# B&R Automation Studio project perfxxl (part 2)

### motorfunc.h
```c
/*
                             *******************
******************************* C HEADER FILE *******************************
**                           *******************                           **
**                                                                         **
** project  : LS JET II                                                    **
** filename : MOTORFUNC.H                                                  **
** version  : 1.02                                                         **
** date     : 24.01.2008                                                   **
**                                                                         **
*****************************************************************************
** Abstract                                                                **
** ========                                                                **
** Declares the functions for motor control functions  	                   **
**                                                                         **
**                                                                         **
** Copyright (c) 2006, Krause-Biagosch GmbH                                **
** All rights reserved.                                                    **
**                                                                         **
*****************************************************************************
VERSION HISTORY:
----------------
Version     : 1.00
Date        : 20.10.2006
Revised by  : Herbert Aden
Description : Original version.

Version     : 1.01
Date        : 12.10.2007
Revised by  : Herbert Aden
Description : signature of MoveToAbsPosition has changed

Version     : 1.02
Date        : 24.01.2008
Revised by  : Herbert Aden
Description : Added define for ANSW0 command

*/

#ifndef _MOTORFUNC_INCLUDED
#define _MOTORFUNC_INCLUDED

/****************************************************************************/
/**                                                                        **/
/**                           INCLUDE FILES                                **/
/**                                                                        **/
/****************************************************************************/
/* NONE */

/****************************************************************************/
/**                                                                        **/
/**                       DEFINITIONS AND MACROS                           **/
/**                                                                        **/
/****************************************************************************/
#define CMDSTRINGLENGTH        (10)
#define DONT_SEND_SPEED        (0L)

#define CMD_RELATIVE_POS            "LR"
#define CMD_ABSOLUTE_POS            "LA"
#define CMD_SPEED                   "SP"
#define CMD_START_MOTION            "M"
#define CMD_CONT_CURRENT            "LCC"
#define CMD_PEAK_CURRENT            "LPC"
#define CMD_STOP                    "V0"
#define CMD_MOVE_AT                 "V"
/* for reference */
#define CMD_HOME                    "HO"
#define CMD_ENABLE                  "EN"
#define CMD_SERIAL                  "SOR0"
#define CMD_ACCELERATION            "AC"
#define CMD_PROPFACT                "POR"
#define CMD_INTFACT                 "I"
#define CMD_NOANSW                  "ANSW0"
#define CMD_COMPATIBLE              "COMPATIBLE1"

#define CMD_GETTEMP                 "TEM"
#define CMD_GETFAULTSTAT            "GFS"

/****************************************************************************/
/**                                                                        **/
/**                      TYPEDEFS AND STRUCTURES                           **/
/**                                                                        **/
/****************************************************************************/
typedef struct
{
	STRING	CmdString[CMDSTRINGLENGTH];  /* command string*/
	DINT	Parameter;          /* Parameter for the command */
	BOOL	UseParameter;       /* if true, the parameter is added to the command
	                             *  else the parameter is ignored
	                             */
	BOOL	UseRefDirection;    /* if true, the ref direction of the motor is used
	                             * to determine the direction of movement
	                             * hence the sign of parameter is irrelevant;
	                             * else the sign is used to determine direction
	                             */
	INT     SendMotor;          /* the motor which shall receive the command*/
	BOOL	Send;               /* the actual send command, stay TRUE until
	                             * sending finished
	                             */
	BOOL	Request;            /* indicates that data is requested from motor */
}SerialCmd_Typ;

/****************************************************************************/
/**                                                                        **/
/**                      EXPORTED VARIABLES                                **/
/**                                                                        **/
/****************************************************************************/
#ifndef _MOTORFUNC_C_SRC
extern _GLOBAL SerialCmd_Typ SerialCmd;
#endif

/****************************************************************************/
/**                                                                        **/
/**                          EXPORTED FUNCTIONS                            **/
/**                                                                        **/
/****************************************************************************/

/****************************************************************************/
/** Send commands to a motor                                                */
/****************************************************************************/
/**
 * Sends commands to a specified motor.
 * Example: Call MotorCmd(1,"LA",TRUE,200000)
 *          will send "1LA200000" to the interface
 *
 * Parameters: UINT  Motor        the motor to which the command is being sent
 *             char *CmdString    the command string (NULL terminated)
 *             BOOL  UseValue     if true, then the value will be added to the
 *                                command
 *             DINT  Value        the value to be added to the command
 *
 * Returns:    OK                 when finished sending
 *             NOT_OK             while waiting for sending
 *
**/
BOOL	SendMotorCmd(const INT pMotor,const char *CmdStr,const BOOL UseValue,const DINT Value);

/****************************************************************************/
/** Check, if a motor is in a certain position window                       */
/****************************************************************************/
/**
 * Checks, if the position of the specified motor is in a specified range
 * (Position window)
 * Example call: PositionOk(1,200000,100)
 *               returns false, as long as the motorposition is <199900
 *                                                           or >200100
 * Parameters: UINT  Motor        the motor to be checked
 *             DINT  Pos          the position where the motor should be
 *             DINT  Deviation    the maximum tolerated deviaition (+/-)
 *
 *
 * Returns:    OK                 if current motor position is in range
 *             NOT_OK             if current motor position is out of range
 *
**/
BOOL	isPositionOk(const INT Motor,DINT Pos,DINT Deviation)/*@modifies nothing@*/;

/****************************************************************************/
/** Check, if a motor is below a certain position                           */
/****************************************************************************/
/**
 * Checks, if the position of the specified motor is below a specified position
 * ATTENTION: Does not work, if actual position has a different sign than the
 *            given max position! May only be used with all positive or all negative
 *            values. E.g. if the atual position is 1000 and we test for -1000 the
 *            function will return true, which wouold be incorrect!!
 *
 * Example call: isPositionLowerThan(1,65000)
 *               returns true, as long as the motorposition is <65000
 *
 * Parameters: UINT  Motor        the motor to be checked
 *             DINT  Pos          the position below which the motor should be
 *
 * Returns:    OK                 if current motor position is lower than
 *                                checkvalue
 *             NOT_OK             if current motor position is higher than or
 *                                equal to checkvalue
 *
**/
BOOL	isPositionLowerThan(const INT Motor,DINT Pos);

/****************************************************************************/
/** Check, if a motor is above a certain position                           */
/****************************************************************************/
/**
 * Checks, if the position of the specified motor is above a specified position
 * ATTENTION: Does not work, if actual position has a different sign than the
 *            given max position! May only be used with all positive or all negative
 *            values. E.g. if the atual position is 1000 and we test for -1000 the
 *            function will return true, which wouold be incorrect!!
 *
 * Example call: isPositionHigherThan(1,65000)
 *               returns true, as long as the motorposition is >65000
 *
 * Parameters: UINT  Motor        the motor to be checked
 *             DINT  Pos          the position below which the motor should be
 *
 * Returns:    OK                 if current motor position is higher than checkvalue
 *             NOT_OK             if current motor position is lower than or equal to
 *                                checkvalue
 *
**/
BOOL	isPositionHigherThan(const INT Motor,DINT Pos);

/****************************************************************************/
/** Request data from a motor                                                */
/****************************************************************************/
/**
 * Requests data from a specified motor.
 * Sets SerialCmd.Request to TRUE, caller must reset this flag after
 * receiving and using the data
 * Example: Call RequestMotorData(1,"TEM")
 *          will send "1TEM" to the interface
 *
 * Parameters: UINT  Motor        the motor to which the command is being sent
 *             char *CmdString    the command string (NULL terminated)
 *
 * Returns:    OK                 when finished sending
 *             NOT_OK             while waiting for sending
 *
**/
BOOL	RequestMotorData(const INT pMotor,const char *CmdString);

/****************************************************************************/
/** Check position of paper remove vertical                                **/
/****************************************************************************/
/**
 * Checks, if the position of the paper remove is in a specified range
 * (Position window)
 * Function is required because PerfoXXL has 2 motors for paper rem. vert.
 *
 * Parameters: DINT  Pos          the position where the motor should be
 *             DINT  Deviation    the maximum tolerated deviaition (+/-)
 *
 *
 * Returns:    OK                 if paper remove vert. position is in range
 *             NOT_OK             if paper remove vert. position is out of range
 *
 * uses        isPositionOk from this module
 *
**/
BOOL	isPapRemVerticalOk(BOOL Config,DINT Pos,UDINT MaxDeviation);

/****************************************************************************/
/* send commands to paper remove vertical */
/****************************************************************************/
/**
 * Sends commands to paper remove vertical.
 * Function is required because PerfoXXL has 2 motors for paper rem. vert.
 *
 * Parameters: char *CmdString    the command string (NULL terminated)
 *             BOOL  UseValue     if true, then the value will be added to the
 *                                command
 *             DINT  Value        the value to be added to the command
 *
 * Returns:    OK                 when finished sending
 *             NOT_OK             while waiting for sending
 *
**/
BOOL	PapRemVerticalCmd(BOOL Config,char *CmdString,BOOL UseValue,DINT Value);

/****************************************************************************/
/* move motor to an absolute position and wait for motion to start */
/****************************************************************************/
/**
 * implements a sequence to send commands to a specified motor to move to an
 * given absolute position at a given speed.
 * The caller must provide a pointer to an USINT variable that will hold the
 * current internal state of the function
 * ATTENTION
 * The function must be called cyclic until it returns OK
 * it returns TRUE only once, as soon as the motion started, then the caller must
 * stop calling, otherwise the motion will start again
 *
 *
 * Parameters: int pMotor         the motor to move
 *             DINT Pos           the position to move to
 *             DINT Speed         the speed of the motion
 *             USINT *pStep       pointer to a USINT var that holds the current step of the
 *                                internal sequence
 *
 * Special parameter values:      -if Speed has the value DONT_SEND_SPEED the speed command
 *                                 will be suppressed and thus one cycle can be saved
 *                                -if all 3 parameters are 0 then the sequence will be reset
 *                                 caller should do this, if the calling sequence is stopped
 *                                 and therefore the function ist no longer called
 *
 * Returns:    TRUE                when motion started
 *             FALSE               during sending
 *
**/
BOOL  MoveToAbsPosition(INT pMotor, DINT Pos, DINT Speed, USINT *pStep);

/****************************************************************************/
/* move motor to an relative position without waiting for motion to start */
/****************************************************************************/
BOOL  MoveToRelPosition(INT pMotor, DINT Pos, DINT Speed, USINT *pStep);

#endif /*_MOTORFUNC_INCLUDED*/

/****************************************************************************/
/**                                                                        **/
/**                                 EOF                                    **/
/**                                                                        **/
/****************************************************************************/
```

### udp.h
```c
/*
                             *******************
******************************* C HEADER FILE *******************************
**                           *******************                           **
**                                                                         **
** project  : X-Jet                                                        **
** filename : UDP.H                                                        **
** version  : 1.00                                                         **
** date     : 08.08.2008                                                   **
**                                                                         **
*****************************************************************************
** Abstract                                                                **
** ========                                                                **
** structs, variables and functions for udp interface to TiffBlaster       **
**                                                                         **
**                                                                         **
** Copyright (c) 2008, Krause-Biagosch GmbH                                **
** All rights reserved.                                                    **
**                                                                         **
*****************************************************************************
VERSION HISTORY:
----------------
Version     : 1.00
Date        : 08.08.2008
Revised by  : Herbert Aden
Description : Original version.

*/

#ifndef _UDP_H
#define _UDP_H

/****************************************************************************/
/**                                                                        **/
/**                           INCLUDE FILES                                **/
/**                                                                        **/
/****************************************************************************/
#include <string.h>
#include <asstring.h>
#include <asudp.h>
#include <bur/plctypes.h>
#include <convert.h>
#include <standard.h>
#include "glob_var.h"
#include "in_out.h"

/****************************************************************************/
/**                                                                        **/
/**                       DEFINITIONS AND MACROS                           **/
/**                                                                        **/
/****************************************************************************/
#define SENDBUFSIZE (400)
#define RCVBUFSIZE (200)
#define DEBUGSTRSIZE (80)

#define INVALIDVALUE (999999999)
#define SEND_OK (1)
#define SEND_BUFFER_FULL (2)
#define SEND_INVALID_PLATETYPE1 (3)
#define SEND_INVALID_PLATETYPE2 (4)
#define SEND_NO_ID (5)
#define SEND_PLATE_NOT_LOADED (6)
#define SEND_MACHINE_NOT_STARTED (7)
#define SEND_WAIT (8)

#define MAXTOKENLENGTH 200
#define MAXTOKENS 20

/****************************************************************************/
/**                                                                        **/
/**                      TYPEDEFS AND STRUCTURES                           **/
/**                                                                        **/
/****************************************************************************/

/****************************************************************************/
/**                                                                        **/
/**                PROJECT GLOBAL VARIABLES                                **/
/**                                                                        **/
/****************************************************************************/
_GLOBAL STRING  RemoteIP[20];
_GLOBAL BOOL	saveRemoteIP;
_GLOBAL BOOL    SendMessageRequest;
_GLOBAL BOOL    SendWarningRequest;
_GLOBAL BOOL    gAbfrageOK,gAbfrageCancel;
_GLOBAL BOOL    gClearLinePressed;

/****************************************************************************/
/**                                                                        **/
/**                          EXPORTED FUNCTIONS                            **/
/**                                                                        **/
/****************************************************************************/
#ifndef _UDP_C
extern    void                init_UDP(void);
extern    void                cyclic_UDP(void);
#endif
/****************************************************************************/
/**                                                                        **/
/**                      EXPORTED VARIABLES                                **/
/**                                                                        **/
/****************************************************************************/
#ifndef _UDP_C
extern    SINT                buffer[SENDBUFSIZE];
extern    UINT                counter;

#else
/****************************************************************************/
/**                                                                        **/
/**                      TASK-LOCAL VARIABLES                              **/
/**                                                                        **/
/****************************************************************************/
_LOCAL    UdpOpen_typ         UDPopen_1,UDPopen_Rcv;
_LOCAL    UdpSend_typ         UDPsend_1;
_LOCAL    UdpRecv_typ         UDPreceive_1;
_LOCAL    UdpClose_typ        UDPclose_1;

_LOCAL    SINT                buffer[SENDBUFSIZE];
_LOCAL    UINT                counter;

_LOCAL    UINT                UDPStep;
_LOCAL    UINT                CounterMax;
_LOCAL    UINT                remotePort;
_LOCAL    SINT                receivebuffer[RCVBUFSIZE];
_LOCAL    UINT                UDPRcvStep;
_LOCAL    STRING              DebugRecStr[DEBUGSTRSIZE];
_LOCAL    STRING              DebugSendStr[DEBUGSTRSIZE];
_LOCAL    UINT                SendStatusInterval;

/****************************************************************************/
/**                                                                        **/
/**                      MODULE-LOCAL VARIABLES                            **/
/**                                                                        **/
/****************************************************************************/
static    TON_10ms_typ        StatusRequestTimer,StatusRequestTimeout;
static    BOOL                SendStatusRequest;
static    BOOL                SendJetStartOK,SendJetStopOK,
                              SendJetRefOK,SendJetControlvoltageOK,SendStepwedgeOK,
                              SendBluefinStartOK,SendBluefinStopOK,
                              SendBluefinControlvoltageOK;
static    USINT               SendJobAnswer,SendJobStates,SendTestAnswer;

static    R_TRIG_typ          MachineOnlineEdgeR,MachineOfflineEdgeR;
static    STRING              tmpID[MAXTOKENLENGTH];
#endif

/****************************************************************************/
/**                                                                        **/
/**                    MODULE-LOCAL VARIABLES                              **/
/**                                                                        **/
/****************************************************************************/
#ifdef _UDP_C
#endif

#endif
/****************************************************************************/
/**                                                                        **/
/**                                 EOF                                    **/
/**                                                                        **/
/****************************************************************************/
```

### Global.typ
```iecst
TYPE
	CANIOcmd_typ : 	STRUCT
		busnr : USINT;
		nodenr : USINT;
		cmd : UDINT;
		res : UDINT;
		status : UINT;
		initcnt : UDINT;
		fcb_ptr : UDINT;
		fcb_cnt : UDINT;
		tiotick : UDINT;
		node_ptr : UDINT;
		local_flag : USINT;
		first_flag : USINT;
		state : USINT;
		pp_ix : USINT;
		enable : BOOL;
	END_STRUCT;
	Command : 	STRUCT
		code : USINT;
		comcode : USINT;
		param1 : USINT;
		param2 : USINT;
		data1 : USINT;
		data2 : USINT;
		data3 : USINT;
		data4 : USINT;
	END_STRUCT;
	EGMPreWashParam_Type : 	STRUCT
		ReplenishingMode : UINT;
		ReplenishmentPerSqm : REAL;
		ReplenishmentPerPlate : REAL;
		ReplenishmentIntervall : UINT;
		PumpMlPerSec : REAL;
		MinPumpOnTime : UINT;
	END_STRUCT;
	EGMPreWash_Type : 	STRUCT
		TankFull : BOOL;
		Pump : BOOL;
		Valve : BOOL;
		HeatingOn : BOOL;
		LevelNotInRange : USINT;
		RealTemperature : INT;
		Auto : BOOL;
		PumpCmd : BOOL;
	END_STRUCT;
	Modules_typ : 	STRUCT
		name : STRING[19];
		info : MoVerStruc_typ;
	END_STRUCT;
	fiLOCAL_OBJ : 	STRUCT
		StateMan : UINT;
		ErrMan : UINT;
		Init : UDINT;
	END_STRUCT;
END_TYPE
```

### Global.var
```iecst
VAR RETAIN
	dummy : ARRAY[0..39] OF USINT;
END_VAR
```

### Program Logical/ip_srv_c (ANSIC, version 1.20.0) - TCP IP Server für zykl. Datenaustausch

#### ip_srv_c.c
```c
#ifdef _DEFAULT_INCLUDES
	#include <AsDefault.h>
#endif
/***************************************************************************/
/*                                                                         */
/* Datei:    ip_srv_c.c                                                    */
/*                                                                         */
/* Autor:    Stefan Hebel / B&R Technisches Büro Nord                      */
/*                                                                         */
/* Abstrakt: Diese Task wartet darauf, daß sich ein TCP-IP Client am ein-  */
/*           gestellten Port anzumelden. Wenn die Verbindung hergestellt   */
/*           worden ist, wartet der Servar auf Daten vom Client. Nachdem   */
/*           Daten erfolgreich empfangen wurden, werden die eigenen Daten  */
/*           gesendet.Nach einem Timeout wird der Port geschlossen und es  */
/*           wird versucht, die Verbindung wieder neu aufzubauen.          */
/*                                                                         */
/* Datum:    11.Aug.2002      letzte Änderungen: 11.Aug.2002 / Heb         */
/*                                                                         */

/*	1.00	xx.xx.xx	  	erstes release			HA		*/
/*	1.10	05.x2.x4	  	bei Befehl 14 wird jetzt auch der Status mitgeschickt		HA		*/
/*							abschaltbar via Kompatibilitätsflag */
/*	1.20	18.09.06	  			*/
/*		 - mehr Sicherheit beim Telnet Server (Längenprüfung der übertragenen strings*/
/*		   besonders beim Einzelzeichen Empfang via telnet konnte man vorher sehr leicht das PP*/
/*		   zum Absturz bringen*/
/*		 - Server ist jetzt nicht mehr case-sensitive und kennt bye, quit und exit um die Verbindung zu trennen */

/***************************************************************************/

/***** Include-Files: *****/
#include <bur/plc.h>
#include <bur/plctypes.h>
#include <Ethernet.h>
#include <string.h>
#include <ctype.h>
#include "asstring.h"
#include "glob_var.h"
#include "in_out.h"
#include "egmglob_var.h"

/***** Variablen-/Konstantendeklaration: *****/
/* Anwendungsspezifische Konstanten: */
#define TCP_IP_PORT		2000				/* Port für Kommunikation */
#define SEND_BUFFER_LEN	150					/* Buffer-Länge für das Senden */
#define RECV_BUFFER_LEN	150					/* Empfangs-Buffer Länge */
#define TIMEOUT			200					/* Abbruch nach TIMEOUT * Zykluszeit Sek.*/
#define	RCVTIMEOUT		200
#define MAXCLIENTS		4
#define	LIVEBYTECNT		160

/* sonstige Konstanten */
#define TCP_IP_OK			0
#define TCP_IP_NO_RCV_DATA	27211
#define TCP_IP_BUSY		65535

#define OPEN_PORT			0
#define WAIT_OPEN_PORT		1
#define SEND_DATA			2
#define WAIT_SEND_DATA		3
#define RECV_DATA			4
#define WAIT_RECV_DATA		5
#define CLOSE_PORT			6
#define WAIT_CLOSE_PORT		7

#define MAXFILENAMELENGTH	32

typedef struct {
	REAL		XPosMm;
	DINT		MotorPos[16];
	REAL		MotorPosMm[16];
	USINT		MotorTemp[16];
	USINT		MotorStatus[16][5];
	USINT		AlarmList[64];
	USINT		Input[16];
	USINT		Output[16];
	USINT		SequenceSteps[16];
	USINT		Trolleys[2];
	USINT		PlateTypes[2];
	USINT		PlateCount[2];
	USINT		MachineStatusBusy;
	USINT		MachineStatusError;
	USINT		MachineStatusStandby;
	USINT		EGMStatus;
	USINT		VCPStatus;
	USINT		TrolleyOpen;
	USINT		PanoramaAdapter;
	USINT		ParameterChanged;
	USINT		PlateAtFeeder;
	USINT		PlateAtShuttle;
	USINT		PlateInDropPosition;
	USINT		PlateAdjusted;
	USINT		PlateAtDeloader;
	USINT		PlateOnConveyorbelt;
	UDINT		PlatesPerHour;
} TSendData;

TSendData	SendData;
_GLOBAL DINT LastStatus;
_GLOBAL	USINT	MotorTemp[MAXMOTORS];
_GLOBAL	STRING	MotorFaultStatus[MAXMOTORS][5];

/* Strukturen fuer Ethernet-Libraray-Funktionen */
_LOCAL	TCPserv_typ			TCP_Server[MAXCLIENTS];
_LOCAL	TCPrecv_typ			TCP_Recv[MAXCLIENTS];
_LOCAL	TCPsend_typ			TCP_Send[MAXCLIENTS];
_LOCAL	TCPclose_typ		TCP_Close[MAXCLIENTS];

/* Variablen: */
SINT	SendBuffer[MAXCLIENTS][SEND_BUFFER_LEN];
SINT	RecvBuffer[MAXCLIENTS][RECV_BUFFER_LEN];
SINT	RecvData[MAXCLIENTS][RECV_BUFFER_LEN];

_LOCAL	SINT	Step[MAXCLIENTS];
_LOCAL	UINT	SendTimeout;
_LOCAL	UINT	RcvLength;
_LOCAL	USINT	LiveByteCnt;
_LOCAL	UINT	ConnectionInvisible;

_LOCAL USINT	tmp[20],test[100];

int CurrentClient,Status,parse;
_LOCAL USINT Count[MAXCLIENTS];

/*HA 23.10.03 V1.67 send laserpower to TiffBlaster if a value is entered (even if it didn't change) */
/*therefore SendLP must be GLOBAL*/
_GLOBAL 	BOOL	SendYOffset,SendLP,SendOSCommand;

_LOCAL	USINT	TimeoutCounter,SendYOffsetStep,SendLPStep,BeamStep,TBShutdownStep,
				SendOSCommandStep;
		UINT	SendYOffsetTimeout,SendLPTimeout,BeamTimeout,OSTimeout;
int i,j,SendCounter,RcvTimeout;
REAL	OldYOffset;
UDINT	OldPower;
_LOCAL int	tmplength;

char pt_tmp[10];
_LOCAL	USINT SendDataCnt[MAXCLIENTS];
BOOL NoAnswer,CloseConnection[MAXCLIENTS];

BOOL SendBData[MAXCLIENTS];
BOOL OldTBVersion;

_GLOBAL USINT *TmpPtr;
_GLOBAL BOOL	PutTmpDataToSRAM;
_LOCAL	BOOL	LoadParamFile,ReadActive;
int LoadParamFileClient;

_GLOBAL	STRING FileIOName[MAXFILENAMELENGTH];
_GLOBAL	STRING	FileType[5];
_GLOBAL	UDINT *FileIOData;
_GLOBAL	UDINT	FileIOLength;
_GLOBAL	BOOL	WriteFileCmd,ReadFileCmd,DeleteFileCmd,WriteFileOK,ReadFileOK,DeleteFileOK,
				FileNotExisting,ReadDirCmd,ReadDirOK,NoDisk;

void StatusToSendBuffer(void)
{
	int i;
/*HA V1.50 send state to TB*/
				strcpy(SendBuffer[0],"ST");
				if (!BUSY && !ERROR && STANDBY)
					strcat(SendBuffer[0],"1");
				else
				if (BUSY && !ERROR && !STANDBY)
					strcat(SendBuffer[0],"2");
				else
				if (!BUSY && ERROR && !STANDBY)
					strcat(SendBuffer[0],"3");
				else
					strcat(SendBuffer[0],"0");

				if ( StatusEGM1 && StatusEGM2 )
					strcat(SendBuffer[0],"0");
				else
					strcat(SendBuffer[0],"1");

				if ( !VCP )
					strcat(SendBuffer[0],"0");
				else
					strcat(SendBuffer[0],"1");

/*erstmal nullen rein*/
					strcat(SendBuffer[0],"0000000000000000000");

/*left trolley*/

				if (GlobalParameter.TrolleyLeft != 0)
				{
					tmplength = itoa((UDINT)(GlobalParameter.TrolleyLeft),(UDINT) &tmp[0]);
					SendBuffer[0][5] = '0';
					SendBuffer[0][6] = '0';
					if(tmplength==1)
						SendBuffer[0][6] = tmp[0];
					else
					{
						SendBuffer[0][5] = tmp[0];
						SendBuffer[0][6] = tmp[1];
					}
/*left platetype*/
					tmplength = itoa((UDINT)(Trolleys[GlobalParameter.TrolleyLeft].PlateType),(UDINT) &tmp[0]);
					SendBuffer[0][9] = '0';
					SendBuffer[0][10] = '0';
					if(tmplength==1)
						SendBuffer[0][10] = tmp[0];
					else
					{
						SendBuffer[0][9] = tmp[0];
						SendBuffer[0][10] = tmp[1];
					}
/*left platestack*/
					tmplength = itoa((UDINT)(Trolleys[GlobalParameter.TrolleyLeft].PlatesLeft),(UDINT) &tmp[0]);
					SendBuffer[0][13] = '0';
					SendBuffer[0][14] = '0';
					SendBuffer[0][15] = '0';
					if(tmplength <= 3 && tmplength > 0)
					{
						for(i=1;i<=tmplength;i++)
							SendBuffer[0][(15+1)-i] = tmp[tmplength-i];
					}
					else
					{
						SendBuffer[0][13] = '9';
						SendBuffer[0][14] = '9';
						SendBuffer[0][15] = '9';
					}

				}
				else	/*no left trolley*/
				{
					SendBuffer[0][5] = '9';
					SendBuffer[0][6] = '9';
					SendBuffer[0][9] = '9';
					SendBuffer[0][10] = '9';
					SendBuffer[0][13] = '9';
					SendBuffer[0][14] = '9';
					SendBuffer[0][15] = '9';
				}

				if (GlobalParameter.TrolleyRight != 0)
				{
					tmplength = itoa((UDINT)(GlobalParameter.TrolleyRight),(UDINT) &tmp[0]);
					SendBuffer[0][7] = '0';
					SendBuffer[0][8] = '0';
					if(tmplength==1)
						SendBuffer[0][8] = tmp[0];
					else
					{
						SendBuffer[0][7] = tmp[0];
						SendBuffer[0][8] = tmp[1];
					}
/*right platetype*/
					tmplength = itoa((UDINT)(Trolleys[GlobalParameter.TrolleyRight].PlateType),(UDINT) &tmp[0]);
					SendBuffer[0][11] = '0';
					SendBuffer[0][12] = '0';
					if(tmplength==1)
						SendBuffer[0][12] = tmp[0];
					else
					{
						SendBuffer[0][11] = tmp[0];
						SendBuffer[0][12] = tmp[1];
					}
/*right platestack*/
					tmplength = itoa((UDINT)(Trolleys[GlobalParameter.TrolleyRight].PlatesLeft),(UDINT) &tmp[0]);
					SendBuffer[0][16] = '0';
					SendBuffer[0][17] = '0';
					SendBuffer[0][18] = '0';
					if(tmplength <= 3 && tmplength > 0)
					{
						for(i=1;i<=tmplength;i++)
							SendBuffer[0][(18+1)-i] = tmp[tmplength-i];
					}
					else
					{
						SendBuffer[0][16] = '9';
						SendBuffer[0][17] = '9';
						SendBuffer[0][18] = '9';
					}
				}
				else
/* no right trolley: left trolley with 2 stacks?*/
				{
					SendBuffer[0][7] = '9';
					SendBuffer[0][8] = '9';

					if (GlobalParameter.TrolleyLeft != 0)
					{
						if (Trolleys[GlobalParameter.TrolleyLeft].Double && Trolleys[GlobalParameter.TrolleyLeft].RightStack)
						{
							tmplength = itoa((UDINT)(Trolleys[GlobalParameter.TrolleyLeft].PlateType),(UDINT) &tmp[0]);
							SendBuffer[0][11] = '0';
							SendBuffer[0][12] = '0';
							if(tmplength==1)
								SendBuffer[0][12] = tmp[0];
							else
							{
								SendBuffer[0][11] = tmp[0];
								SendBuffer[0][12] = tmp[1];
							}
/*right platestack*/
							tmplength = itoa((UDINT)(Trolleys[GlobalParameter.TrolleyLeft].PlatesRight),(UDINT) &tmp[0]);
							SendBuffer[0][16] = '0';
							SendBuffer[0][17] = '0';
							SendBuffer[0][18] = '0';
							if(tmplength <= 3 && tmplength > 0)
							{
								for(i=1;i<=tmplength;i++)
									SendBuffer[0][(18+1)-i] = tmp[tmplength-i];
							}
							else
							{
								SendBuffer[0][16] = '9';
								SendBuffer[0][17] = '9';
								SendBuffer[0][18] = '9';
							}
						}
						else  /* no right trolley and no right stack*/
						{
							SendBuffer[0][7] = '9';
							SendBuffer[0][8] = '9';
							SendBuffer[0][11] = '9';
							SendBuffer[0][12] = '9';
							SendBuffer[0][16] = '9';
							SendBuffer[0][17] = '9';
							SendBuffer[0][18] = '9';
						}
					}
				}

				if (/*PanoramaAdapter*/ ManualMode)
				{
					SendBuffer[0][19] = 'P';
/*Plate Type from Pano Input*/
					tmplength = itoa((UDINT)(PlateType),(UDINT) &tmp[0]);
					SendBuffer[0][9] = '0';
					SendBuffer[0][10] = '0';
					SendBuffer[0][11] = '0';
					SendBuffer[0][12] = '0';
					if(tmplength==1)
					{
						SendBuffer[0][10] = tmp[0];
						SendBuffer[0][12] = tmp[0];
					}
					else
					{
						SendBuffer[0][9] = tmp[0];
						SendBuffer[0][10] = tmp[1];
						SendBuffer[0][11] = tmp[0];
						SendBuffer[0][12] = tmp[1];
					}
				}
				else
					SendBuffer[0][19] = ' ';

				if(TrolleyOpen)
					SendBuffer[0][20] = 'O';
				else
					SendBuffer[0][20] = 'C';

/*Alarmbitfield übertragen*/
				for(i=0;i<MAXALARMS;i++)
				{
					SendBuffer[0][21+i] = AlarmBitField[i]+48;
				}
/* HA 28.07.05 zusätzliche Info an Netlink: Wieviele Platten im System und welcher Typ*/
				SendBuffer[0][21+MAXALARMS] =  '0';
				SendBuffer[0][21+MAXALARMS+1] =  '0';
				tmplength = itoa((UDINT)(UnexposedPlatesInSystem),(UDINT) &tmp[0]);
				if(tmplength==1)
				{
					SendBuffer[0][21+MAXALARMS] =  tmp[0];
					if (/*PanoramaAdapter*/ ManualMode)
						tmplength = itoa((UDINT)(PlateType),(UDINT) &tmp[0]);
					else
					/* q&d für Performance */
						tmplength = itoa((UDINT)(Trolleys[GlobalParameter.TrolleyLeft].PlateType),(UDINT) &tmp[0]);

					if(tmplength==1)
						SendBuffer[0][21+MAXALARMS+1] =  tmp[0];
				}

				TCP_Send[0].buflng = 21+MAXALARMS;
}

/***** INIT FUNKTION *******************************************************/
_INIT void init (void)
{
	int i;
	CurrentClient = 1;
	/* Initialisierung der TCP-IP Datenstrukturen: */

	for(i = 0;i<MAXCLIENTS;i++)
	{
		SendBData[i] = 0;
		SendDataCnt[i] = 0;
		/* TCP-IP Client: */
		TCP_Server[i].enable	= TRUE;
		TCP_Server[i].porta	= TCP_IP_PORT+i;

		/* TCP-IP Client Senden: */
		TCP_Send[i].enable		= TRUE;
		TCP_Send[i].buffer		= (UDINT)&SendBuffer[i][0];
		TCP_Send[i].buflng		= SEND_BUFFER_LEN;

		/* TCP-IP Client Empfangen: */
		TCP_Recv[i].enable		= TRUE;
		TCP_Recv[i].buffer		= (UDINT)&RecvBuffer[i][0];
		TCP_Recv[i].mxbuflng	= RECV_BUFFER_LEN;

		/* TCP-IP Client schließen */
		TCP_Close[i].enable	= TRUE;

		Step[i] = OPEN_PORT;
		Count[i] = 0;
		CloseConnection[i] = 0;
	}

	OldYOffset =0.0;
	OldPower =0;
	SendCounter=0;
	OldTBVersion = 0;
	LoadParamFile = 0;

} /* Ende Funktion _INIT void init (void) */

/***** ZYKLISCHE FUNKTION **************************************************/
_CYCLIC void cyclic (void)
{
	/***** Öffnen des Ports ************************************************/
	if (Step[0] == OPEN_PORT)
	{
		/* 1. Aufruf der Funktion */
		TCPserv (&TCP_Server[0]);
		Step[0] = WAIT_OPEN_PORT;
	}
	if (Step[0] == WAIT_OPEN_PORT)
	{
		/* Status prüfen: */
		if (TCP_Server[0].status == TCP_IP_OK)
		{
			/* Port geöffnet */
			/* Identifier zuordnen ... */
			TCP_Send[0].cident = TCP_Server[0].cident;
			TCP_Recv[0].cident = TCP_Server[0].cident;
			TCP_Close[0].cident = TCP_Server[0].cident;
			/* ... und zum nächsten Schritt gehen */
			Step[0] = RECV_DATA;
			TCPConnected = 1;
			ConnectionInvisible = 0;
			SendYOffset = 1;
			SendLP = 1;
			AlarmBitField[24] = 0;
		}
		else
		{
			/* Funktion erneut aufrufen */
			TCPserv (&TCP_Server[0]);
			TCPConnected = 0;
			ConnectionInvisible = 1;
		}
	} /* if (Step == WAIT_OPEN_PORT) */

/**************************************************************/
/*  Y-OFFSET */
/**************************************************************/

/*detect changed Offset*/
	if(PlateParameter.YOffset != OldYOffset && TCPConnected )
	{
		OldYOffset = PlateParameter.YOffset;
		SendYOffset = 1;
	}

	switch (SendYOffsetStep)
	{
		case 0:
		{
			if(SendYOffset && TCPConnected )
			{
				if( PlateParameter.YOffset>=0.00 && PlateParameter.YOffset<=999.99)
					SendYOffsetStep = 5;
				else
					SendYOffset = 0;
			}
			break;
		}
		case 5:
		{
			if(TCPSendCmd == 0)
			{
				strcpy(TCPCmd,"YO");
				tmplength = itoa((UDINT)(PlateParameter.YOffset *100),(UDINT) &tmp[0]);
/*fill the string with zeros to get fixed 5 digits*/
				for(i=0;i< 5-tmplength;i++)
				{
					TCPCmd[2+i] = '0';
					TCPCmd[2+i+1] = 0;
				}
				tmp[5] = 0; /*safety!*/
				strcat(TCPCmd,tmp);
				TCPSendCmd = 1;
				SendYOffsetStep = 8;
			}
			SendYOffsetTimeout = 0;
			break;
		}
		case 8:
		{
			if( !TCPRcvFlag)
			{
				SendYOffsetTimeout++;
				if(SendYOffsetTimeout>150)
				{
					SendCounter++;
					if(SendCounter < 5)
						SendYOffsetStep = 5;
					else
					{
					/*ERROR*/
						SendYOffsetStep = 0;
						SendYOffset = 0;
						SendCounter = 0;
						AlarmBitField[24] = 1;
					}
				}
				break;
			}

			AlarmBitField[24] = 0;
/*check for YOOK*/
			if( !strcmp(TCPAnswer,"YOOK") )
			{
				TCPRcvFlag = 0;
				SendYOffsetStep = 0;
				SendYOffset = 0;
				SendYOffsetTimeout = 0;
				SendCounter = 0;
			}

			break;
		}
	} /*switch*/

/**************************************************************/
/*  BEAM ON/OFF*/
/**************************************************************/
	switch (BeamStep)
	{
		case 0:
		{
			if( (BeamON || BeamOFF) && TCPConnected )
			{
				if(BeamON && BeamOFF) BeamON = 0;
				BeamStep = 5;
			}
			break;
		}
		case 5:
		{
			if(TCPSendCmd == 0)
			{
				if(BeamON)
					strcpy(TCPCmd,"43=ON");
				if(BeamOFF)
					strcpy(TCPCmd,"43=OFF");
				TCPSendCmd = 1;
				BeamStep = 8;
			}
			BeamTimeout = 0;
			break;
		}
		case 8:
		{
			if( !TCPRcvFlag)
			{
				BeamTimeout++;
				if(BeamTimeout>150)
				{
					SendCounter++;
					if(SendCounter < 5)
						BeamStep = 5;
					else
					{
					/*ERROR*/
						BeamStep = 0;
						BeamON = 0;
						BeamOFF = 0;
						SendCounter = 0;
						AlarmBitField[24] = 1;
					}
				}
				break;
			}

			AlarmBitField[24] = 0;
/*check for answer*/
			if( ( !strcmp(TCPAnswer,"SSH1") && BeamON )
			||  ( !strcmp(TCPAnswer,"SSH0") && BeamOFF ) )
			{
				TCPRcvFlag = 0;
				BeamStep = 0;
				BeamON = 0;
				BeamOFF = 0;
				BeamTimeout = 0;
				SendCounter = 0;
			}

			break;
		}
	} /*switch*/

/**************************************************************/
/*  TIFF Blaster shutdown*/
/**************************************************************/
	switch (TBShutdownStep)
	{
		case 0:
		{
/*safety*/
			if( !TCPConnected )
				TBShutdown = 0;

			if( (TBShutdown) && TCPConnected )
			{
				TBShutdownStep = 5;
			}
			break;
		}
		case 5:
		{
			if(TCPSendCmd == 0)
			{
				strcpy(TCPCmd,"SD");
				TCPSendCmd = 1;
				TBShutdownStep = 0;
				TBShutdown = 0;
			}
			break;
		}
	} /*switch*/

/**************************************************************/
/*  TIFF Blaster: Open Beam shutter */
/* V1.36 */
/**************************************************************/
	switch (SendOSCommandStep)
	{
		case 0:
		{
/*safety*/
			if( !TCPConnected )
				SendOSCommand = 0;

			if( (SendOSCommand) && TCPConnected )
			{
				SendOSCommandStep = 5;
			}
			break;
		}
		case 5:
		{
			if(TCPSendCmd == 0)
			{
				strcpy(TCPCmd,"OS");
				TCPSendCmd = 1;
				OSTimeout = 0;
				SendOSCommandStep = 8;
			}
			break;
		}
		case 8:
		{
			if( !TCPRcvFlag)
			{
				OSTimeout++;
				if(OSTimeout>150)
				{
					SendCounter++;
					if(SendCounter < 5)
						SendOSCommandStep = 5;
					else
					{
					/*ERROR*/
						SendOSCommandStep = 0;
						SendOSCommand = 0;
						SendCounter = 0;
						OSTimeout = 0;
						AlarmBitField[24] = 1;
					}
				}
				break;
			}

			AlarmBitField[24] = 0;
/*check for answer*/
			if( !strcmp(TCPAnswer,"OSOK"))
			{
				TCPRcvFlag = 0;
				SendOSCommandStep = 0;
				SendOSCommand = 0;
				SendCounter = 0;
				OSTimeout = 0;
				SendCounter = 0;
			}

			break;
		}

	} /*switch*/

/**************************************************************/
/*  LASERPOWER*/
/**************************************************************/

/*detect changed Laserpower*/
	if(GlobalParameter.RealLaserPower != OldPower && TCPConnected )
	{
		OldPower = GlobalParameter.RealLaserPower;
		SendLP = 1;
	}

	switch (SendLPStep)
	{
		case 0:
		{
			if(SendLP && TCPConnected )
			{
				if( GlobalParameter.RealLaserPower > 0 && GlobalParameter.RealLaserPower <= 1000)
				{
					SendLPStep = 1;
					AlarmBitField[31] = 0;
					AlarmBitField[32] = 0;
				}
				else
					SendLP = 0;
			}
			break;
		}

/*HA 28.07.04 V1.81 Tiffblaster Version abfragen*/
		case 1:
		{
			if(TCPSendCmd == 0)
			{
				strcpy(TCPCmd,"VER?");
				TCPSendCmd = 1;
				SendLPStep = 2;
			}
			SendLPTimeout = 0;
			break;
		}

		case 2:
		{
			if( !TCPRcvFlag)
			{
				SendLPTimeout++;
				if(SendLPTimeout>150)
				{
					SendCounter++;
					if(SendCounter < 5)
						SendLPStep = 1;
					else
					{
					/*ERROR, no answer: maybe old version, go ahead...*/
						SendLPStep = 5;
						SendLPTimeout = 0;
						SendCounter = 0;
						OldTBVersion = 1;
						SendLP = 0;
					}
				}
				break;
			}

/*Antwort empfangen, Auswertung*/
			AlarmBitField[24] = 0;
			TCPRcvFlag = 0;
			SendLPStep = 5;
			SendLPTimeout = 0;
			SendCounter = 0;

/*check for "Failure"->old version */
			if( !strcmp(TCPAnswer,"Failure") )
				OldTBVersion = 1;
			else
				OldTBVersion = 0;

			break;
		}

		case 5:
		{
			if(TCPSendCmd == 0)
			{
				if (OldTBVersion)
				{
					strcpy(TCPCmd,"LP");
					tmplength = itoa((UDINT)(GlobalParameter.LaserPower),(UDINT) &tmp[0]);
/*fill the string with zeros to get fixed 3 digits*/
					for(i=0;i< 3-tmplength;i++)
					{
						TCPCmd[2+i] = '0';
						TCPCmd[2+i+1] = 0;
					}
					tmp[3] = 0; /*safety!*/
					strcat(TCPCmd,tmp);
				}
				else /*neue Version 4 stellig*/
				{
					strcpy(TCPCmd,"LX");
					tmplength = itoa((UDINT)(GlobalParameter.RealLaserPower),(UDINT) &tmp[0]);
/*fill the string with zeros to get fixed 4 digits*/
					for(i=0;i< 4-tmplength;i++)
					{
						TCPCmd[2+i] = '0';
						TCPCmd[2+i+1] = 0;
					}
					tmp[4] = 0; /*safety!*/
					strcat(TCPCmd,tmp);
				}
				TCPSendCmd = 1;
				SendLPStep = 8;
			}
			SendLPTimeout = 0;
			break;
		}
		case 8:
		{
			if( !TCPRcvFlag)
			{
				SendLPTimeout++;
				if(SendLPTimeout>150)
				{
					SendCounter++;
					if(SendCounter < 5)
						SendLPStep = 5;
					else
					{
					/*ERROR*/
						SendLPStep = 0;
						SendLP = 0;
						SendCounter = 0;
						AlarmBitField[24] = 1;
					}
				}
				break;
			}

			AlarmBitField[24] = 0;
/*check for LPOK*/
			if( !strcmp(TCPAnswer,"LPOK") )
			{
				TCPRcvFlag = 0;
				SendLPStep = 10;
				SendLPTimeout = 0;
				SendCounter = 0;
			}

			break;
		}

/* HA 22.01.04 V1.74 New step to check for answer (result)*/
		case 10:
		{
/*HA 09.02.04 V1.75 Kompatibilitätsflag prüfen*/
			if ( GlobalParameter.UseOldTiffBlaster )
			{
				SendLPStep = 0;
				SendLP = 0;
				SendCounter = 0;
				break;
			}

			if( !TCPRcvFlag)
			{
				SendLPTimeout++;
				if(SendLPTimeout>12000)
				{
					/*ERROR timeout*/
					SendLPStep = 0;
					SendLP = 0;
					SendCounter = 0;
				}
				break;
			}

			AlarmBitField[24] = 0;
/*check for LPREADY*/
			if( !strcmp(TCPAnswer,"LPREADY") )
			{
				TCPRcvFlag = 0;
				SendLPStep = 0;
				SendLP = 0;
				SendLPTimeout = 0;
				SendCounter = 0;
			}
			else
/*check for LPFAILED*/
			if( !strcmp(TCPAnswer,"LPFAILED") )
			{
				TCPRcvFlag = 0;
				SendLPStep = 0;
				SendLP = 0;
				SendLPTimeout = 0;
				SendCounter = 0;
				AlarmBitField[31] = 1;
/* Laser power setting failed: error message */
				AbfrageText1 = 0;
				AbfrageText2 = 54;
				AbfrageText3 = 0;

				if(wBildAktuell != MESSAGEPIC )
					OrgBild = wBildAktuell;
				wBildNeu = MESSAGEPIC;
				AbfrageOK = 0;
				AbfrageCancel = 0;
				IgnoreButtons = 1;
				OK_CancelButtonInv = 1;
				OK_ButtonInv = 0;
				AbfrageIcon = CAUTION;
			}

			break;
		}	/*case 10*/

	} /*switch*/

	/***** Daten Empfangen *************************************************/
	if (TCPConnected)
	{
		TCPrecv (&TCP_Recv[0]);
		/* Status prüfen: */
		if (TCP_Recv[0].status == TCP_IP_OK)
		{
			if(TCP_Recv[0].rxbuflng == 0) /*CLOSE von Gegenstelle*/
			{
				Step[0] = CLOSE_PORT;
			}
			else	/* Daten empfangen -> auswerten*/
			{
/*check for LPERROR*/
				if( !memcmp(RecvBuffer[0],"LPERROR",7) )
				{
					START = 0;
					AlarmBitField[32] = 1;
	/* Laser power error message */
					AbfrageText1 = 0;
					AbfrageText2 = 55;
					AbfrageText3 = 0;

					if(wBildAktuell != MESSAGEPIC )
						OrgBild = wBildAktuell;
					wBildNeu = MESSAGEPIC;
					AbfrageOK = 0;
					AbfrageCancel = 0;
					IgnoreButtons = 1;
					OK_CancelButtonInv = 1;
					OK_ButtonInv = 0;
					AbfrageIcon = CAUTION;
				}
				else
				{
					TCPRcvFlag = 1;
					strcpy(TCPAnswer,RecvBuffer[0]);
					RcvLength = TCP_Recv[0].rxbuflng;
					TCPAnswer[RcvLength-1] = 0;
				}
			}
		}
/*Wenn keiner das  receive flag löscht, nach Zeit selbst löschen*/
		if(TCPRcvFlag)
		{
			RcvTimeout++;
			if(RcvTimeout > RCVTIMEOUT)
			{
				RcvTimeout=0;
				TCPRcvFlag = 0;
			}
		}
	}

	/***** Daten Senden ****************************************************/
	/***** Lebenszeichen Senden *******************************************/
	if(TCPConnected)
	{
		if(TCPSendCmd != 0)
		{
			if(TCPSendCmd == 2) /*Livebyte*/
			{
				StatusToSendBuffer();
			}
			else
			{
				if ( !strcmp(TCPCmd,"14") && !GlobalParameter.UseOldTiffBlaster ) /*soll 14 geschickt werden?*/
				{
					StatusToSendBuffer();
					SendBuffer[0][0] = '1';
					SendBuffer[0][1] = '4';
				}
				else
				if ( !strcmp(TCPCmd,"15"))  /*soll 15 geschickt werden?*/
				{
					StatusToSendBuffer();
					SendBuffer[0][0] = '1';
					SendBuffer[0][1] = '5';
				}
				else
				{
					memcpy(SendBuffer[0],TCPCmd,strlen(TCPCmd));
					TCP_Send[0].buflng = strlen(TCPCmd);
				}
			}

			TCPsend (&TCP_Send[0]);
			/* Status prüfen: */
			if (TCP_Send[0].status == TCP_IP_OK)
			{
			/* Senden war OK */
				TCPSendCmd = 0;
				SendTimeout = 0;
			}
			SendTimeout++;
			LiveByteCnt = 0;
			if(SendTimeout > TIMEOUT)
			{
				Step[0] = CLOSE_PORT;
				TCPSendCmd = 0;
				SendTimeout = 0;
				TCPConnected = 0;
				ConnectionInvisible = 1;
			}
		}
/*no sending? send livebyte */
		else
		{
			LiveByteCnt++;
			if(LiveByteCnt > LIVEBYTECNT)
			{
				if(TCPSendCmd == 0)
				{
					TCPSendCmd = 2;
					LiveByteCnt = 0;
				}
			}
		}
	}
	else /*no connection: reset send Cmd*/
		TCPSendCmd = 0;

	/***** Port schließen **************************************************/
	if (Step[0] == CLOSE_PORT)
	{
		TCPConnected = 0;
		ConnectionInvisible = 1;
		TCPclose (&TCP_Close[0]);
		Step[0] = WAIT_CLOSE_PORT;
	}
	if (Step[0] == WAIT_CLOSE_PORT)
	{
		/* Status prüfen: */
		if (TCP_Close[0].status == TCP_IP_OK)
		{
			/* Port geschlossen, neu öffnen: */
			Step[0] = OPEN_PORT;
		}
		else
		{
			/* Funktion erneut aufrufen */
			TCPclose (&TCP_Close[0]);
		}
	} /* if (Step == WAIT_CLOSE_PORT) */

/***************************************************************************/
/***************************************************************************/
/*		weitere Clients bedienen                                           */
/*                                                                         */

			SendData.XPosMm = FU.aktuellePosition_mm;
			for(i=0;i<16;i++)
			{
				SendData.MotorPos[i] = Motors[i].Position;
				SendData.MotorPosMm[i] = Motors[i].Position_mm;
				SendData.MotorTemp[i] = MotorTemp[i];
				for(j=0;j<4;j++)
					SendData.MotorStatus[i][j] = MotorFaultStatus[i][j];
				SendData.MotorStatus[i][4] = 0;
			}

			for(i=0;i<MAXALARMS;i++)
				SendData.AlarmList[i] = AlarmBitField[i];

			SendData.Input[0] = BeltLoose;
			SendData.Input[1] = 0;
			SendData.Input[2] = TrolleyCodeSensor;
			SendData.Input[3] = In_ConveyorBeltSensor[0];
			SendData.Input[4] = 0;
			SendData.Input[5] = 0;
			SendData.Input[6] = 0;
			SendData.Input[7] = 0;
			SendData.Input[8] = InEGM1;
			SendData.Input[9] = InEGM2;
			SendData.Input[10] = VCP;
			SendData.Input[11] = CoverLockOK;
			SendData.Input[12] = DoorsOK;
			SendData.Input[13] = 0;
			SendData.Input[14] = 0;
			SendData.Input[15] = 0;
/*
			SendData.Output[0] = out0;
			SendData.Output[1] = out1;
			SendData.Output[2] = out2;
			SendData.Output[3] = out3;
			SendData.Output[4] = out4;
			SendData.Output[5] = out5;
			SendData.Output[6] = out6;
			SendData.Output[7] = out7;
			SendData.Output[8] = out8;
			SendData.Output[9] = out9;
			SendData.Output[10] = out10;
			SendData.Output[11] = out11;
			SendData.Output[12] = out12;
			SendData.Output[13] = out13;
			SendData.Output[14] = out14;
			SendData.Output[15] = out15;
*/
			for(i=0;i<10;i++)
				SendData.SequenceSteps[i] = SequenceSteps[i];
/*HA 11.05.04 V1.77*/
			SendData.SequenceSteps[15] = CurrentStack;
/*
	SeqenceSteps[0]	PaperRemove
	SeqenceSteps[1]	Feeder
	SeqenceSteps[2]	Shuttle
	SeqenceSteps[3]	Adjust
	SeqenceSteps[4]	Expose
	SeqenceSteps[5]	Deload
	SeqenceSteps[6]	TrolleyOpen
	SeqenceSteps[7]	TrolleyClose
	SeqenceSteps[8]	Reference
*/

/*Status data*/
			SendData.MachineStatusBusy = BUSY;
			SendData.MachineStatusError = ERROR;
			SendData.MachineStatusStandby = STANDBY;
			SendData.EGMStatus = !(StatusEGM1 && StatusEGM2);
			SendData.VCPStatus = !VCP;
			SendData.Trolleys[0] = GlobalParameter.TrolleyLeft;
			SendData.Trolleys[1] = GlobalParameter.TrolleyRight;

			if (GlobalParameter.TrolleyLeft != 0)
			{
				SendData.PlateTypes[0] = Trolleys[GlobalParameter.TrolleyLeft].PlateType;
				SendData.PlateCount[0] = Trolleys[GlobalParameter.TrolleyLeft].PlatesLeft;
			}
			else
			{
				SendData.PlateTypes[0] = 0;
				SendData.PlateCount[0] = 0;
			}

			if (GlobalParameter.TrolleyRight != 0)
			{
				SendData.PlateTypes[1] = Trolleys[GlobalParameter.TrolleyRight].PlateType;
				SendData.PlateCount[1] = Trolleys[GlobalParameter.TrolleyRight].PlatesLeft;
			}
			else
			{
/*2 stacks in double size trolley ?*/
				if (GlobalParameter.TrolleyLeft != 0)
				{
					if (Trolleys[GlobalParameter.TrolleyLeft].Double && Trolleys[GlobalParameter.TrolleyLeft].RightStack)
					{
						SendData.PlateTypes[1] = Trolleys[GlobalParameter.TrolleyLeft].PlateType;
						SendData.PlateCount[1] = Trolleys[GlobalParameter.TrolleyLeft].PlatesRight;
					}
					else
					{
						SendData.PlateTypes[1] = 0;
						SendData.PlateCount[1] = 0;
					}
				}
			}

			if (PanoramaAdapter)
			{
				SendData.PanoramaAdapter = 1;
				SendData.PlateTypes[0] = SendData.PlateTypes[1] = PlateType;
			}
			else
				SendData.PanoramaAdapter = 0;

			if(TrolleyOpen)
				SendData.TrolleyOpen = 1;
			else
				SendData.TrolleyOpen = 0;

			if (ParameterChanged)
				SendData.ParameterChanged = 1;
			ParameterChanged = 0;

			SendData.PlateAtFeeder = PlateAtFeeder.present;
			SendData.PlateAtShuttle = 0;
			SendData.PlateInDropPosition = 0;
			SendData.PlateAdjusted = AdjustReady;
			SendData.PlateAtDeloader = PlateAtDeloader.present;
			SendData.PlateOnConveyorbelt = PlateOnConveyorBelt.present;
			SendData.PlatesPerHour = PlatesPerHour;

	for(CurrentClient = 1;CurrentClient<MAXCLIENTS;CurrentClient++)
	{
	/***** Öffnen des Ports ************************************************/
		if (Step[CurrentClient] == OPEN_PORT)
		{
 			CloseConnection[CurrentClient] = 0;
			/* 1. Aufruf der Funktion */
			TCPserv (&TCP_Server[CurrentClient]);
			/* Status prüfen: */
			if (TCP_Server[CurrentClient].status == TCP_IP_OK)
			{
				/* Port geöffnet */
				/* Identifier zuordnen ... */
				TCP_Send[CurrentClient].cident = TCP_Server[CurrentClient].cident;
				TCP_Recv[CurrentClient].cident = TCP_Server[CurrentClient].cident;
				TCP_Close[CurrentClient].cident = TCP_Server[CurrentClient].cident;
				/* ... und zum nächsten Schritt gehen */
				Step[CurrentClient] = RECV_DATA;
			}
		} /* if (Step == WAIT_OPEN_PORT) */

	/***** Daten Empfangen *************************************************/
		if (Step[CurrentClient] == RECV_DATA)
		{
			TCPrecv (&TCP_Recv[CurrentClient]);
			/* Status prüfen: */
			if (TCP_Recv[CurrentClient].status == TCP_IP_OK)
			{
				if(TCP_Recv[CurrentClient].rxbuflng == 0) /*CLOSE von Gegenstelle*/
				{
					Step[CurrentClient] = CLOSE_PORT;
					Count[CurrentClient] = 0;
				}
				else	/* Daten empfangen -> auswerten*/
				{
					parse = 0;
					/*einzelne Zeichen (via telnet)*/
					if(TCP_Recv[CurrentClient].rxbuflng < 3)
					{
						RecvData[CurrentClient][Count[CurrentClient]] = RecvBuffer[CurrentClient][0];
						Count[CurrentClient]++;
/* safety !*/
						if (Count[CurrentClient] >= RECV_BUFFER_LEN )
						{
							strcpy(SendBuffer[CurrentClient],"HEY! \a\aSTOP SENDING!!");
							Step[CurrentClient] = SEND_DATA;
							TCP_Send[CurrentClient].buffer		= (UDINT)&SendBuffer[CurrentClient];
							TCP_Send[CurrentClient].buflng = strlen(SendBuffer[CurrentClient]);
							Count[CurrentClient] = 0;
							parse = 0;
						}
						else
						if( RecvBuffer[CurrentClient][0] == 10 || RecvBuffer[CurrentClient][0] == 13 )
						{
							RecvData[CurrentClient][Count[CurrentClient]] = 0;
							parse = 1;
						}
					}
					else
					{
						memcpy(RecvData[CurrentClient],RecvBuffer[CurrentClient],TCP_Recv[CurrentClient].rxbuflng);
						Count[CurrentClient] = TCP_Recv[CurrentClient].rxbuflng;
						parse = 1;
					}

					if(parse)
					{
						i=0;
						while ( RecvData[CurrentClient][i] != 0 )
						{
							RecvData[CurrentClient][i] = toupper( RecvData[CurrentClient][i] );
							i++;
						}
						RecvData[CurrentClient][Count[CurrentClient]-1] = 0;
						if( strncmp(RecvData[CurrentClient],"STATUS",6) == 0 )
						{
							if(BUSY)
								strcpy(SendBuffer[CurrentClient],"ST=BUSY\r\n");
							else if(ERROR)
									strcpy(SendBuffer[CurrentClient],"ST=ERROR\r\n");
								else if(STANDBY)
										strcpy(SendBuffer[CurrentClient],"ST=READY\r\n");
						}
						else
						if( strncmp(RecvData[CurrentClient],"SPEED",5) == 0 )
						{
							strcpy(SendBuffer[CurrentClient],"SPEED=");
							itoa(PlatesPerHour,(UDINT) &tmp[0]);
							strcat(SendBuffer[CurrentClient],tmp);
							strcat(SendBuffer[CurrentClient],"\r\n");
						}
						else
						if( strncmp(RecvData[CurrentClient],"TROLLEY",7) == 0 )
						{
							if(GlobalParameter.TrolleyLeft != 0)
							{
								strcpy(SendBuffer[CurrentClient],"LEFT=");
								itoa(Trolleys[GlobalParameter.TrolleyLeft].PlatesLeft,(UDINT) &tmp[0]);
								strcat(SendBuffer[CurrentClient],tmp);
								if(Trolleys[GlobalParameter.TrolleyLeft].Double)
								{
									strcat(SendBuffer[CurrentClient]," RIGHT=");
									itoa(Trolleys[GlobalParameter.TrolleyLeft].PlatesRight,(UDINT) &tmp[0]);
									strcat(SendBuffer[CurrentClient],tmp);
								}
							}
							else
							{
								strcpy(SendBuffer[CurrentClient],"");
							}
							if(GlobalParameter.TrolleyRight != 0)
							{
								if(GlobalParameter.TrolleyLeft != 0)
									strcat(SendBuffer[CurrentClient]," RIGHT=");
								else
									strcat(SendBuffer[CurrentClient],"RIGHT=");
								itoa(Trolleys[GlobalParameter.TrolleyRight].PlatesLeft,(UDINT) &tmp[0]);
								strcat(SendBuffer[CurrentClient],tmp);
							}
							if(GlobalParameter.TrolleyLeft == 0 && GlobalParameter.TrolleyRight == 0)
								strcpy(SendBuffer[CurrentClient],"NO TROLLEY");
							strcat(SendBuffer[CurrentClient],"\r\n");
						}
						else
/*noch nicht wirklich gut, sobald ein client dieses command schickt, wird das flag für alle */
/* global zurückgesetzt, besser: binäre sendedaten auch als array*/
						if (strncmp(RecvData[CurrentClient],"RESETPARAMCHANGED",17) == 0)
						{
							SendData.ParameterChanged = 0;
							NoAnswer = 1;
						}
						else
/* Load a specific parameter file */
/* syntax: LOADPARAMFILE BLAH\r\n   ohne Endung! */
						if (strncmp(RecvData[CurrentClient],"LOADPARAMFILE",13) == 0)
						{
							LoadParamFile = 1;
							LoadParamFileClient = CurrentClient;
							strcpy(FileIOName,&RecvData[CurrentClient][14]);
							FileIOName[strlen(FileIOName)-1] = 0; /*CRLF entfernen*/
							strcpy(SendBuffer[CurrentClient],"LOADPARAMFILE OK\r\n");
						}
						else
						if (strncmp(RecvData[CurrentClient],"BYE",3) == 0
						||	strncmp(RecvData[CurrentClient],"QUIT",4) == 0
						||	strncmp(RecvData[CurrentClient],"EXIT",4) == 0)
						{
							strcpy(SendBuffer[CurrentClient],"Good bye, cu next time...\r\n");
							CloseConnection[CurrentClient] = 1;
						}
						else
						{
							memcpy(tmp,RecvData[CurrentClient],10);
							tmp[10] = 0;
							if( strcmp(tmp,"LASERPOWER") == 0 )
							{
								/*new power to set?*/
								if(Count[CurrentClient] > 11 && RecvData[CurrentClient][10]=='=')
								{
									i=11;
									while (isdigit(RecvData[CurrentClient][i]) && i<Count[CurrentClient]) i++;
									if (i>11)
									{
										memcpy(tmp,&RecvData[CurrentClient][11],i-11);
										GlobalParameter.RealLaserPower = atoi((UDINT) &tmp);
									}
								}
								strcpy(SendBuffer[CurrentClient],"LASERPOWER=");
								itoa(GlobalParameter.RealLaserPower,(UDINT) &tmp[0]);
								strcat(SendBuffer[CurrentClient],tmp);
								strcat(SendBuffer[CurrentClient],"\r\n");
							}
							else
								strcpy(SendBuffer[CurrentClient],"unknown command\r\n");
						}
						Step[CurrentClient] = SEND_DATA;
						TCP_Send[CurrentClient].buffer		= (UDINT)&SendBuffer[CurrentClient];
						TCP_Send[CurrentClient].buflng = strlen(SendBuffer[CurrentClient]);
						Count[CurrentClient] = 0;
						parse = 0;
					}
					SendDataCnt[CurrentClient]=0;
				}
			}
			else
			{
/*nothing received: ok, send binary data*/
				if (TCP_Recv[CurrentClient].status == TCP_IP_NO_RCV_DATA)
				{
					SendDataCnt[CurrentClient]++;
					if( SendDataCnt[CurrentClient] >= 10)
					{
						SendDataCnt[CurrentClient] = 0;
						SendBData[CurrentClient] = 1;
					}
				}
			}
		}

/************** senden ****************************/

		if ( SendBData[CurrentClient] )
		{
			SendBData[CurrentClient] = 0;

			TCP_Send[CurrentClient].buffer		= (UDINT)&SendData;
			TCP_Send[CurrentClient].buflng		= sizeof (SendData);
			Step[CurrentClient] = SEND_DATA;
		}

		if (Step[CurrentClient] == SEND_DATA)
		{

			TCPsend (&TCP_Send[CurrentClient]);
			/* Status prüfen: */
			if (TCP_Send[CurrentClient].status == TCP_IP_OK)
			{
				/* Senden war OK */
				if (CloseConnection[CurrentClient])
					Step[CurrentClient] = CLOSE_PORT;
				else
					Step[CurrentClient] = RECV_DATA;
				CloseConnection[CurrentClient] = 0;
			}
			else
			if ( (TCP_Send[CurrentClient].status != TCP_IP_BUSY)  &&
				(TCP_Send[CurrentClient].status != ERR_ETH_NET_SLOW)
					)
			{
				LastStatus = TCP_Send[CurrentClient].status;
				if (TCP_Send[CurrentClient].status==14896)
					Step[CurrentClient] = RECV_DATA;
				else
					Step[CurrentClient] = CLOSE_PORT;
			}
		}

	/***** Port schließen **************************************************/
		if (Step[CurrentClient] == CLOSE_PORT)
		{
			TCPclose (&TCP_Close[CurrentClient]);
			/* Status prüfen: */
			if (TCP_Close[CurrentClient].status == TCP_IP_OK)
			{
				/* Port geschlossen, neu öffnen: */
				Step[CurrentClient] = OPEN_PORT;
			}
		} /* if (Step == WAIT_CLOSE_PORT) */

	} /*for*/

	if (LoadParamFile)
	{
		/*try to load sram from file*/
		FileIOData = (UDINT *) TmpPtr;
#ifdef MODE_BOTH
		FileIOLength = OVERALLSRAMSIZEEBYTES;
		strcpy(FileType,"SA1");
#else
	#ifdef MODE_PERFORMANCE
		FileIOLength = PERFSRAMSIZEBYTES;
		strcpy(FileType,"SA1");
	#else
		#ifdef MODE_BLUEFIN
		FileIOLength = OVERALLSRAMSIZEEBYTES;
		strcpy(FileType,"SA1");
		#endif
	#endif
#endif

		if(!ReadActive)
		{
			ReadActive = 1;
			ReadFileCmd = 1;
			ReadFileOK = 0;
			FileNotExisting = 0;
		}
		else
		{
/*wait for reading ready*/
			if(ReadFileOK)
			{
				LoadParamFile = 0;
				ReadActive = 0;
				ReadFileOK = 0;
				/*save to SRAM*/
				PutTmpDataToSRAM = 1;
				strcpy(SendBuffer[LoadParamFileClient],"PARAM FILE LOADED SUCCESSFULLY!");
				Step[LoadParamFileClient] = SEND_DATA;
				TCP_Send[LoadParamFileClient].buffer		= (UDINT)&SendBuffer[LoadParamFileClient][0];
				TCP_Send[LoadParamFileClient].buflng = strlen(SendBuffer[LoadParamFileClient]);

			}
/*file not existing*/
			if(FileNotExisting)
			{
				LoadParamFile = 0;
				ReadActive = 0;
				ReadFileOK = 0;
				FileNotExisting = 0;
				strcpy(SendBuffer[LoadParamFileClient],"PARAM FILE NOT FOUND!\r\n");
				Step[LoadParamFileClient] = SEND_DATA;
				TCP_Send[LoadParamFileClient].buffer		= (UDINT)&SendBuffer[LoadParamFileClient][0];
				TCP_Send[LoadParamFileClient].buflng = strlen(SendBuffer[LoadParamFileClient]);
			}
		}
	} /*if (loadparamfile)*/

} /* Ende Funktion _CYCLIC void cyclic (void) */

/* ENDE */
```

### Program Logical/sram (ANSIC, version 1.10.0) - Daten in SRAM sichern bzw wieder auslesen
